// TwinCAT 3 PLC project TcIotOcppServer1Plc
// Title: TwinCAT IoT OCPP Server Sample
// Company: Beckhoff Automation GmbH & Co. KG
// ProjectVersion: 1.0.3.0
// ProgramVersion: 3.1.4026.16
// CompilerDefines: VISU_USEPROPERTYINFO
// libraries:
//   Tc2_EtherCAT, * (Beckhoff Automation GmbH)
//   Tc2_Standard, * (Beckhoff Automation GmbH)
//   Tc2_System, * (Beckhoff Automation GmbH)
//   Tc2_Utilities, * (Beckhoff Automation GmbH)
//   Tc3_Module, * (Beckhoff Automation GmbH)
//   Tc3_OCPP, * (Beckhoff Automation GmbH)
//   VisuDialogs, * (System)
//   VisuSymbols, 4.5.0.0 (System)
// project tree:
//   DUTs/ ST_Connector.TcDUT, ST_VisuStation.TcDUT
//   / GlobalTextList.TcGTLO, PlcTask.TcTTO, Visualization Manager.TcVMO (not stored)
//   GVLs/ VAR_OCPP.TcGVL
//   POUs/ FB_SampledValueMeasurands.TcPOU, FB_Server.TcPOU, FB_Station.TcPOU, MAIN.TcPOU
//   POUs/Helper/ F_ChargePointStatusToString.TcPOU, F_TimeFromString.TcPOU
//   VISUs/ Main_Visu.TcVIS, Measurand.TcVIS, Visu_BootNotification.TcVIS, Visu_Connector.TcVIS, Visu_Station.TcVIS
// real-time tasks:
//   TASK PlcTask: cycle T#1ms, priority 20, ADS port 350

CONFIGURATION TcIotOcppServer1Plc
    RESOURCE PLC ON TwinCAT3
        TASK PlcTask(INTERVAL := T#1ms, PRIORITY := 20);
        PROGRAM MAIN WITH PlcTask : MAIN;
    END_RESOURCE
END_CONFIGURATION

// ---- DUTs/ST_Connector.TcDUT
TYPE ST_Connector :
STRUCT
	sIdTag 				: T_OCPP1_IdToken;
	nReservationId 		: UDINT;
	sStartTime 			: STRING(255);
	sAuthorizationStatus : E_OCPP1_AuthorizationStatus;
	sStopTime 			: STRING(255);
	nTransactionID 		: UDINT; 
	nMeterStart 		: UDINT; // Wh
	nMeterStop 			: UDINT; // Wh 
	sChargpointStatus 	: STRING(31); 
END_STRUCT
END_TYPE

// ---- DUTs/ST_VisuStation.TcDUT
TYPE ST_VisuStation :
STRUCT
	sIdent : T_OCPP_Identity; 
	stBoot : ST_OCPP1_ClientBootInfo; 
	aConnector : ARRAY [0 .. Tc3_Ocpp.Param_OCPP.nConnectorCount] OF ST_Connector; 
END_STRUCT
END_TYPE

// ---- GVLs/VAR_OCPP.TcGVL
{attribute 'qualified_only'}
VAR_GLOBAL
	arrAuthList : ARRAY[1..nAuthListMax] OF ST_OCPP1_AuthorizationData := [
		( sIdTag := '1234abcd', stIdTagInfo := ( eStatus := E_OCPP1_AuthorizationStatus.Accepted ) ),
		( sIdTag := 'B45E00EE', stIdTagInfo := ( eStatus := E_OCPP1_AuthorizationStatus.Accepted ) ),
		( sIdTag := 'A46FF2F1', stIdTagInfo := ( eStatus := E_OCPP1_AuthorizationStatus.Accepted ) )
	];

	stServerParam : ST_OCPP1_ServerParam := (
		//nOID := 16#01010010); 	// ObjectID of the TcIotOcpp Client Object (0 to create a new instance).
		nTaskOID 	:= 0, 			// ObjectId of the Task whose shall execute the client (0 to use I/O Idle Task)
		sHost 		:= '0.0.0.0', 	// Defines the server-address by host-name, domain-name or IP-address.
		nPort 		:= 8080, 		// Defines the server-port.
		sPath 		:= 'ocpp', 		// Defines the server-path.
		eAuthMode 	:= E_OCPP1_AuthenticationMode.Basic, 			// Defines an optional authentication-mode.
		eEncryptionMode := E_OCPP_EncryptionMode.None, 				// Defines an optional encryption mode.
		eEncryptionMode := E_OCPP_EncryptionMode.None, 				// Defines an optional encryption mode.
		eEncryptionProt := E_OCPP_EncryptionProtocol.TLSv1p2, 		// Defines the encryption protocol.
		sCaFile 	:= '%TC_TARGETPATH%\Certificates\CA.crt', 		// Certificate of the certificate authority (CA) as filename (PEM or DER format).
		sCrtFile 	:= '%TC_TARGETPATH%\Certificates\OCPP.crt', 	// Certificate of the server (public key) as filename (PEM or DER format)
		sKeyFile 	:= '%TC_TARGETPATH%\Certificates\OCPP.key', 	// Key of the server (private key) as filename (PEM or DER format).
		eDebugLevel := E_OCPP_DebugLevel.None, 		// Defines the debug level.
		eTraceLevel := TcTraceLevel.tlWarning); 	// Defines the maximum trace level of ADS log messages	
END_VAR

VAR_GLOBAL CONSTANT
	nAuthListMax : UDINT := 3;
	sIdTag : T_OCPP1_IdToken := '1234abcd';
	nReservationId : UDINT := 1234;
END_VAR

// ---- POUs/MAIN.TcPOU
PROGRAM MAIN
VAR
	fbServer : FB_Server(VAR_OCPP.stServerParam);

	fbStation01 : FB_Station('ChargingStation01', '2f20aa42275837973ed8f3726bb2709e0a9e476da9c42da38ac113de818d0dbf', fbServer); // ChargingStation01:abcdef
	fbStation02 : FB_Station('ChargingStation02', '5c55b2828abee6bb262ed0505d53d0baa947e050825ef00e7d3432b722177480', fbServer); // ChargingStation02:abcdef
	//fbStation03 : FB_Station('ChargingStation03', 'f207afc2a29d076265649b050ff3f6449b03dc6d04620e269a17cb31584a4471', fbServer); // ChargingStation03:abcdef
END_VAR

fbStation01.Execute();
fbStation02.Execute();
fbServer.Execute();

END_PROGRAM

// ---- POUs/FB_Server.TcPOU
FUNCTION_BLOCK FB_Server
VAR_OUTPUT
	bValid : BOOL;
END_VAR
VAR
	_fbServer 	: FB_OCPP1_Server(0);
	// receive
	hStationId 	: UDINT;
	hMessageId 	: T_OCPP_MessageId;
	eAction 	: E_OCPP1_Action;
END_VAR

METHOD Execute : BOOL
bValid := _fbServer.bValid;
IF NOT bValid THEN RETURN; END_IF
END_METHOD

METHOD FB_Init : BOOL
VAR_INPUT
	bInitRetains : BOOL; // if TRUE, the retain variables are initialized (warm start / cold start)
	bInCopyCode : BOOL;  // if TRUE, the instance afterwards gets moved into the copy code (online change)

	stParam : REFERENCE TO ST_OCPP1_ServerParam;
END_VAR
IF bInCopyCode THEN RETURN; END_IF

FB_Init := _fbServer.Init(stParam);
END_METHOD

PROPERTY Server : REFERENCE TO FB_OCPP1_Server
GET
Server REF= _fbServer;
END_GET
END_PROPERTY

END_FUNCTION_BLOCK

// ---- POUs/FB_Station.TcPOU
FUNCTION_BLOCK FB_Station
VAR_OUTPUT
	bValid 			: BOOL;
	bOpen			: BOOL;
	bRecv 			: BOOL;
	bReserved 		: BOOL;
	arrCharging 	: ARRAY[0..Param_OCPP.nConnectorCount] OF BOOL; 
	arrStatus 		: ARRAY[0..Param_OCPP.nConnectorCount] OF E_OCPP1_ChargePointStatus;
	arrMeasurands 	: ARRAY[0..Param_OCPP.nConnectorCount] OF FB_SampledValueMeasurands;
END_VAR
VAR
	_fbStation 		: FB_OCPP1_Station('', '', 0);
	_bRecvBoot 		: BOOL := TRUE;
	_bRecvStatus 	: BOOL := TRUE;
	_bRecvMeter 	: BOOL := TRUE;
	_nSendState 	: UDINT;
	_hMessageId 	: T_OCPP_MessageId;
	_eTriggerStatus : E_OCPP1_TriggerMessageStatus;
	
	_stVisu 		: ST_VisuStation;
	_arrRemoteStart	: ARRAY[0..Param_OCPP.nConnectorCount] OF BOOL; 
	_arrRemoteStop	: ARRAY[0..Param_OCPP.nConnectorCount] OF BOOL; 
END_VAR
VAR PERSISTENT
	_nTransactionId		: UDINT;
	_arrTransactionId 	: ARRAY[0..Param_OCPP.nConnectorCount] OF UDINT;
	_arrMeterStart 		: ARRAY[0..Param_OCPP.nConnectorCount] OF UDINT; // [Wh]
	_arrMeterStop 		: ARRAY[0..Param_OCPP.nConnectorCount] OF UDINT; // [Wh]
END_VAR

METHOD ActionHistory : BOOL
VAR_INPUT
	eAction : E_OCPP1_Action;
END_VAR
VAR_STAT
	arrHistory : ARRAY[1..cnCount] OF E_OCPP1_Action;
END_VAR
VAR CONSTANT
	cnCount : UDINT := 100;
END_VAR
MEMMOVE(ADR(arrHistory[2]), ADR(arrHistory[1]), SIZEOF(arrHistory[1]) * (cnCount - 1));
arrHistory[1] := eAction;
END_METHOD

METHOD Authorize : BOOL
VAR_IN_OUT CONSTANT
	sId : T_OCPP1_IdToken;
END_VAR
VAR
	nIdx : UDINT;
END_VAR
FOR nIdx := 1 TO VAR_OCPP.nAuthListMax DO
	IF VAR_OCPP.arrAuthList[nIdx].sIdTag = '' THEN
		RETURN;
	END_IF
	IF VAR_OCPP.arrAuthList[nIdx].sIdTag = sId THEN
		Authorize := (VAR_OCPP.arrAuthList[nIdx].stIdTagInfo.eStatus = E_OCPP1_AuthorizationStatus.Accepted);
		RETURN;
	END_IF
END_FOR
END_METHOD

METHOD Execute : BOOL
VAR_STAT
	hMessageId : T_OCPP_MessageId;
	eAction : E_OCPP1_Action;
	eSendState : E_OCPP1_Action;
	nConnectorId : UDINT; 
END_VAR
VAR
	nIdx : UDINT; 
END_VAR
bValid := _fbStation.bValid;
IF NOT bValid THEN RETURN; END_IF

IF NOT bOpen AND_THEN _fbStation.IsConnected THEN
	bOpen := TRUE;
	bRecv := TRUE;
ELSIF bOpen AND_THEN NOT _fbStation.IsConnected THEN
	bOpen := FALSE;
END_IF

IF _fbStation.PollRequest(eAction => eAction, hMessageId => hMessageId) THEN
	bRecv := TRUE;
	ActionHistory(eAction);
	CASE eAction OF
		E_OCPP1_Action.BootNotification:
			RecvBootNotification();
		E_OCPP1_Action.Heartbeat:
			RecvHeartbeat();
		E_OCPP1_Action.MeterValues:
			RecvMeterValues();
		E_OCPP1_Action.StatusNotification:
			RecvStatusNotification();
		E_OCPP1_Action.Authorize:
			RecvAuthorize();
		E_OCPP1_Action.StartTransaction:
			RecvStartTransaction();
		E_OCPP1_Action.StopTransaction:
			RecvStopTransaction();
		E_OCPP1_Action.DiagnosticsStatusNotification:
			RecvDiagnosticsStatusNotification();
		E_OCPP1_Action.FirmwareStatusNotification:
			RecvFirmwareStatusNotification();
		E_OCPP1_Action.DataTransfer:
			RecvDataTransfer();
		E_OCPP1_Action.SecurityEventNotification:
			RecvSecurityEventNotification();
	ELSE
		_fbStation.RespError(hMessageId, eAction, E_OCPP1_Error.NotImplemented);
	END_CASE
END_IF

// RemoteStart/-Stop from Visu
FOR nIdx := 1 TO Param_OCPP.nConnectorCount DO 
	IF _arrRemoteStart[nIdx] THEN 
		_nSendState := E_OCPP1_Action.RemoteStartTransaction;
		_arrRemoteStart[nIdx] := FALSE; 
		nConnectorId := nIdx; 
	ELSIF _arrRemoteStop[nIdx] THEN 
		_nSendState := E_OCPP1_Action.RemoteStopTransaction;
		_arrRemoteStop[nIdx] := FALSE; 
		nConnectorId := nIdx;
	END_IF
	
	IF nConnectorId = 2 OR NOT bOpen THEN 
		_nSendState := 0;	// Connector not implementet or not connectet
	END_IF
END_FOR

CASE _nSendState OF
	0: // idle
		bRecv := FALSE;
	1:
		IF bRecv THEN
			IF _bRecvBoot THEN
				_bRecvBoot := FALSE;
				_nSendState := 10;
			ELSIF _bRecvStatus THEN
				_bRecvStatus := FALSE;
				_nSendState := 20;
			ELSIF _bRecvMeter THEN
				_bRecvMeter := FALSE;
				_nSendState := 30;
			END_IF
			bRecv := FALSE;
		END_IF
	10: // BootNotification
		IF _fbStation.SendTriggerMessage(eRequestedMessage:= E_OCPP1_MessageTrigger.BootNotification, nConnectorId:= 0, eStatus=> _eTriggerStatus) THEN
			_nSendState := 0;
		END_IF
	20: // StatusNotification
		IF _fbStation.SendTriggerMessage(eRequestedMessage:= E_OCPP1_MessageTrigger.StatusNotification, nConnectorId:= 0, eStatus=> _eTriggerStatus) THEN
			IF _eTriggerStatus = E_OCPP1_TriggerMessageStatus.Accepted THEN
				_nSendState := 21;
			ELSE
				arrStatus[0] := E_OCPP1_ChargePointStatus.Unavailable;
				_nSendState := 0;
			END_IF
		END_IF
	21: // StatusNotification
		IF _fbStation.SendTriggerMessage(eRequestedMessage:= E_OCPP1_MessageTrigger.StatusNotification, nConnectorId:= 1, eStatus=> _eTriggerStatus) THEN
			IF _eTriggerStatus = E_OCPP1_TriggerMessageStatus.Accepted THEN
				_nSendState := 22;
			ELSE
				arrStatus[1] := E_OCPP1_ChargePointStatus.Unavailable;
				_nSendState := 0;
			END_IF
		END_IF
	22: // StatusNotification
		IF _fbStation.SendTriggerMessage(eRequestedMessage:= E_OCPP1_MessageTrigger.StatusNotification, nConnectorId:= 2, eStatus=> _eTriggerStatus) THEN
			IF _eTriggerStatus = E_OCPP1_TriggerMessageStatus.Accepted THEN
				_nSendState := 0;
			ELSE
				arrStatus[2] := E_OCPP1_ChargePointStatus.Unavailable;
				_nSendState := 0;
			END_IF
		END_IF
	30: // MeterValues
		IF _fbStation.SendTriggerMessage(eRequestedMessage:= E_OCPP1_MessageTrigger.MeterValues, nConnectorId:= 0, eStatus=> _eTriggerStatus) THEN
				_nSendState := 31;
		END_IF
	31: // MeterValues
		IF _fbStation.SendTriggerMessage(eRequestedMessage:= E_OCPP1_MessageTrigger.MeterValues, nConnectorId:= 1, eStatus=> _eTriggerStatus) THEN
			IF _eTriggerStatus = E_OCPP1_TriggerMessageStatus.Accepted THEN
				_nSendState := 32;
			ELSE
				_nSendState := 0;
			END_IF
		END_IF
	32: // MeterValues
		IF _fbStation.SendTriggerMessage(eRequestedMessage:= E_OCPP1_MessageTrigger.MeterValues, nConnectorId:= 2, eStatus=> _eTriggerStatus) THEN
			IF _eTriggerStatus = E_OCPP1_TriggerMessageStatus.Accepted THEN
				_nSendState := 0;
			ELSE
				_nSendState := 0;
			END_IF
		END_IF
	E_OCPP1_Action.RemoteStartTransaction:
		SendRemoteStartTransaction();
	E_OCPP1_Action.RemoteStopTransaction:
		SendRemoteStopTransaction();
	E_OCPP1_Action.ChangeAvailability:
		SendChangeAvailability();
	E_OCPP1_Action.ChangeConfiguration:
		SendChangeConfiguration();
	E_OCPP1_Action.GetConfiguration:
		SendGetConfiguration();
	E_OCPP1_Action.UnlockConnector:
		SendUnlockConnector();
	E_OCPP1_Action.ClearCache:
		SendClearCache();
	E_OCPP1_Action.Reset:
		SendReset();
	E_OCPP1_Action.TriggerMessage:
		SendTriggerMessage();
	E_OCPP1_Action.ReserveNow:
		SendReserveNow();
	E_OCPP1_Action.CancelReservation:
		SendCancelReservation();
	E_OCPP1_Action.SetChargingProfile:
		SendChargingProfile();
	E_OCPP1_Action.GetCompositeSchedule:
		SendGetCompositeSchedule();
	E_OCPP1_Action.ClearChargingProfile:
		SendClearChargingProfile();
	E_OCPP1_Action.GetLocalListVersion:
		SendGetLocalListVersion();
	E_OCPP1_Action.SendLocalList:
		SendLocalList();
	E_OCPP1_Action.GetDiagnostics:
		SendGetDiagnostics();
	E_OCPP1_Action.UpdateFirmware:
		SendUpdateFirmware();
	E_OCPP1_Action.DataTransfer:
		SendDataTransfer();
ELSE
	_nSendState := 0;
END_CASE

IF _nSendState = 0 AND eSendState <> 0 THEN
	_nSendState := eSendState;
	eSendState := 0;
END_IF

FOR nIdx := 1 TO Param_OCPP.nConnectorCount DO 
	IF arrCharging[nIdx] THEN 
		_stVisu.aConnector[nIdx].sStopTime := ''; 
		_stVisu.aConnector[nIdx].nMeterStop := 0; 
	ELSE 
		_stVisu.aConnector[nIdx].nMeterStart := _arrMeterStart[nIdx];
		_stVisu.aConnector[nIdx].nMeterStop := _arrMeterStop[nIdx];
	END_IF
	_stVisu.aConnector[nIdx].nTransactionID := _arrTransactionId[nIdx]; 
	_stVisu.aConnector[nIdx].sChargpointStatus := TO_STRING(arrStatus[nIdx]); 
END_FOR
END_METHOD

METHOD FB_Init : BOOL
VAR_INPUT
	bInitRetains : BOOL; // if TRUE, the retain variables are initialized (warm start / cold start)
	bInCopyCode : BOOL;  // if TRUE, the instance afterwards gets moved into the copy code (online change)

	sIdent : T_OCPP_Identity;
	sAuthHash : T_OCPP_Hash;
	fbServer : REFERENCE TO FB_Server;
END_VAR
IF bInCopyCode THEN RETURN; END_IF
_stVisu.sIdent := sIdent; 
FB_Init := _fbStation.Init(sIdent, sAuthHash, fbServer.Server);
END_METHOD

METHOD RecvAuthorize : BOOL
VAR_STAT
	sIdTag : T_OCPP1_IdToken;
END_VAR
IF _fbStation.RecvAuthorize(hMessageId => _hMessageId, sIdTag => sIdTag) THEN
	IF Authorize(sIdTag) THEN
		_fbStation.RespAuthorize(_hMessageId, eStatus := E_OCPP1_AuthorizationStatus.Accepted);
	ELSE
		_fbStation.RespAuthorize(_hMessageId, eStatus := E_OCPP1_AuthorizationStatus.Invalid);
	END_IF
END_IF
END_METHOD

METHOD RecvBootNotification : BOOL
VAR_STAT
	sModel 				: STRING(31);
	sVendor 			: STRING(31);
	sChargeBoxSerial 	: STRING(31);
	sChargePointSerial 	: STRING(31);
	sFirmwareVersion 	: STRING(63);
	sMeterSerial 		: STRING(31);
	sMeterType 			: STRING(31);
END_VAR
IF _fbStation.RecvBootNotification(hMessageId=> _hMessageId,
	sModel=> sModel,
	sVendor=> sVendor,
	sChargeBoxSerial=> sChargeBoxSerial,
	sChargePointSerial=> sChargePointSerial,
	sFirmwareVersion=> sFirmwareVersion,
	sMeterSerial=> sMeterSerial,
	sMeterType=> sMeterType)
THEN
	_fbStation.RespBootNotification(_hMessageId, eStatus := E_OCPP1_RegistrationStatus.Accepted);
			
	_stVisu.stBoot.sChargePointModel 		:= sModel; 				
	_stVisu.stBoot.sChargePointVendor 		:= sVendor; 			
	_stVisu.stBoot.sChargeBoxSerialNumber 	:= sChargeBoxSerial; 	
	_stVisu.stBoot.sChargePointSerialNumber	:= sChargePointSerial; 	
	_stVisu.stBoot.sFirmwareVersion 		:= sFirmwareVersion;	
	_stVisu.stBoot.sMeterSerialNumber 		:= sMeterSerial; 		
	_stVisu.stBoot.sMeterType 				:= sMeterType; 			
	
	_bRecvBoot := FALSE;
END_IF
END_METHOD

METHOD RecvDataTransfer : BOOL
VAR_STAT
	sVendorId : STRING(255);
	sMessageId : STRING(63);
	sData : T_OCPP1_DataTransferData;
END_VAR
IF _fbStation.RecvDataTransfer(hMessageId => _hMessageId,
	sVendorId=> sVendorId,
	sMessageId=> sMessageId,
	sData := sData)
THEN
	IF sVendorId <> 'Beckhoff Automation' THEN
		_fbStation.RespDataTransfer(_hMessageId, eStatus := E_OCPP1_DataTransferStatus.UnknownVendorId);
	ELSIF sMessageId <> 'DataTransfer' THEN
		_fbStation.RespDataTransfer(_hMessageId, eStatus := E_OCPP1_DataTransferStatus.UnknownMessageId);
	ELSE
		_fbStation.RespDataTransfer(_hMessageId, eStatus := E_OCPP1_DataTransferStatus.Accepted);
	END_IF
END_IF
END_METHOD

METHOD RecvDiagnosticsStatusNotification : BOOL
IF _fbStation.RecvDiagnosticsStatusNotification(hMessageId => _hMessageId) THEN
	_fbStation.RespDiagnosticsStatusNotification(_hMessageId);
END_IF
END_METHOD

METHOD RecvFirmwareStatusNotification : BOOL
IF _fbStation.RecvFirmwareStatusNotification(hMessageId => _hMessageId) THEN
	_fbStation.RespFirmwareStatusNotification(_hMessageId);
END_IF
END_METHOD

METHOD RecvHeartbeat : BOOL
VAR_STAT
	nHeartbeats : UDINT;
END_VAR
IF _fbStation.RecvHeartbeat(hMessageId => _hMessageId) THEN
	nHeartbeats := nHeartbeats + 1;
	_fbStation.RespHeartbeat(_hMessageId);
END_IF
END_METHOD

METHOD RecvMeterValues : BOOL
VAR_STAT
	nConnectorId : UDINT;
	nTransactionId : UDINT;
	nSampleCount : UDINT;
	arrSampleValues : ARRAY[1..Param_OCPP.nSampledValuesMax] OF ST_OCPP1_SampledValue;
END_VAR
IF _fbStation.RecvMeterValue(
	hMessageId => _hMessageId,
	nConnectorId => nConnectorId,
	nTransactionId => nTransactionId,
	nSampleCount => nSampleCount,
	aSampleValues := arrSampleValues)
THEN
	IF nConnectorId >= 0 AND nConnectorId <= Param_OCPP.nConnectorCount THEN
		arrMeasurands[nConnectorId].Update(arrSampleValues);
	END_IF
	_fbStation.RespMeterValue(_hMessageId);
	_bRecvMeter := FALSE;
END_IF
END_METHOD

METHOD RecvSecurityEventNotification : BOOL
VAR_STAT
	nTimestamp : ULINT;
	sType : STRING(63);
	sInfo : STRING(256);
END_VAR
IF _fbStation.RecvSecurityEventNotification(hMessageId => _hMessageId,
	nTimestamp => nTimestamp,
	sType => sType,
	sInfo => sInfo)
THEN
	_fbStation.RespSecurityEventNotification(_hMessageId);
END_IF
END_METHOD

METHOD RecvStartTransaction : BOOL
VAR_STAT
	sIdTag : T_OCPP1_IdToken;
	nConnectorId : UDINT;
	nMeterStart : UDINT;
	nReservationId : UDINT;
	nTimestamp : ULINT;
END_VAR
IF _fbStation.RecvStartTransaction(hMessageId => _hMessageId,
	sIdTag => sIdTag,
	nConnectorId => nConnectorId,
	nMeterStart => nMeterStart,
	nReservationId => nReservationId,
	nTimestamp => nTimestamp)
THEN


	_stVisu.aConnector[nConnectorId].sIdTag := sIdTag; 
	
	IF Authorize(sIdTag) THEN
		IF nConnectorId >= 1 AND nConnectorId <= Param_OCPP.nConnectorCount THEN
			_nTransactionId := _nTransactionId + 1;
			_arrTransactionId[nConnectorId] := _nTransactionId;
			_arrMeterStart[nConnectorId] := nMeterStart;
			_fbStation.RespStartTransaction(_hMessageId, eStatus := E_OCPP1_AuthorizationStatus.Accepted, nTransactionId := _nTransactionId);
			arrCharging[nConnectorId] := TRUE; 
			_stVisu.aConnector[nConnectorId].nReservationId := nReservationId; 
			_stVisu.aConnector[nConnectorId].sStartTime := TO_STRING(FILETIME64_TO_DT(nTimestamp)); 			
			_stVisu.aConnector[nConnectorId].sAuthorizationStatus := E_OCPP1_AuthorizationStatus.Accepted; 
			RETURN;
		END_IF
	END_IF
	_fbStation.RespStartTransaction(_hMessageId, eStatus := E_OCPP1_AuthorizationStatus.Invalid, nTransactionId := 0);
END_IF
END_METHOD

METHOD RecvStatusNotification : BOOL
VAR_STAT
	nConnectorId : UDINT;
	eError : E_OCPP1_ChargePointError;
	eStatus : E_OCPP1_ChargePointStatus;
	nTimestamp : ULINT := 0;
	sInfo : STRING(63) := '';
	sVendorError : STRING(63) := '';
	sVendorId : STRING(255) := '';
END_VAR
IF _fbStation.RecvStatusNotification(hMessageId => _hMessageId,
	nConnectorId => nConnectorId,
	eError => eError,
	eStatus => eStatus,
	nTimestamp => nTimestamp,
	sInfo => sInfo,
	sVendorError => sVendorError,
	sVendorId => sVendorId)
THEN
	IF nConnectorId >= 0 AND nConnectorId <= Param_OCPP.nConnectorCount THEN
		arrStatus[nConnectorId] := eStatus;
		StatusHistory(nConnectorId, eStatus);
		arrCharging[nConnectorId] := (eStatus = E_OCPP1_ChargePointStatus.Charging);
		bReserved := (eStatus = E_OCPP1_ChargePointStatus.Reserved);
	END_IF
	_fbStation.RespStatusNotification(_hMessageId);
	_bRecvStatus := FALSE;
END_IF
END_METHOD

METHOD RecvStopTransaction : BOOL
VAR_STAT
	sIdTag : T_OCPP1_IdToken;
	nTransactionId : UDINT;
	nConnectorId : UDINT;
	nMeterStop : UDINT;
	nTimestamp : ULINT;
	eReason : E_OCPP1_Reason;
END_VAR
VAR
	nIdx : UDINT;
END_VAR
IF _fbStation.RecvStopTransaction(hMessageId => _hMessageId,
	sIdTag => sIdTag,
	nTransactionId => nTransactionId,
	nConnectorId => nConnectorId,
	nMeterStop => nMeterStop,
	nTimestamp => nTimestamp,
	eReason => eReason)
THEN
	IF sIdTag = '' OR_ELSE Authorize(sIdTag) THEN
		IF nConnectorId >= 1 AND nConnectorId <= Param_OCPP.nConnectorCount THEN
			_arrTransactionId[nConnectorId] := 0;
			_arrMeterStop[nConnectorId] := nMeterStop;
			_fbStation.RespStopTransaction(_hMessageId, eStatus := E_OCPP1_AuthorizationStatus.Accepted);
			arrCharging[nConnectorId] := FALSE; 
			
			_stVisu.aConnector[nConnectorId].sStopTime := TO_STRING(FILETIME64_TO_DT(nTimestamp));
			RETURN;
		END_IF
		FOR nIdx := 1 TO Param_OCPP.nConnectorCount DO
			IF _arrTransactionId[nIdx] = nTransactionId THEN
				_arrTransactionId[nIdx] := 0;
				_arrMeterStop[nIdx] := nMeterStop;
				_fbStation.RespStopTransaction(_hMessageId, eStatus := E_OCPP1_AuthorizationStatus.Accepted);
				arrCharging[nIdx] := FALSE; 
				
				_stVisu.aConnector[nIdx].sStopTime := TO_STRING(FILETIME64_TO_DT(nTimestamp)); 
				RETURN;
 			END_IF
		END_FOR
	END_IF
	_fbStation.RespStopTransaction(_hMessageId, eStatus := E_OCPP1_AuthorizationStatus.Invalid);
END_IF
END_METHOD

METHOD SendCancelReservation : BOOL
VAR_STAT
	nReservationId : UDINT := VAR_OCPP.nReservationId;
	eStatus : E_OCPP1_CancelReservationStatus;
END_VAR
IF _fbStation.SendCancelReservation(nReservationId:= nReservationId, eStatus=> eStatus) THEN
	bReserved := (eStatus <> E_OCPP1_CancelReservationStatus.Accepted);
	_nSendState := 0;
END_IF
END_METHOD

METHOD SendChangeAvailability : BOOL
VAR_STAT
	nConnectorId : UDINT := 1;
	eType : E_OCPP1_AvailabilityType;
	eStatus : E_OCPP1_AvailabilityStatus;
END_VAR
IF eType = E_OCPP1_AvailabilityType.None THEN
	IF arrStatus[1] = E_OCPP1_ChargePointStatus.Unavailable THEN
		eType := E_OCPP1_AvailabilityType.Operative;
	ELSE
		eType := E_OCPP1_AvailabilityType.Inoperative;
	END_IF
END_IF
IF _fbStation.SendChangeAvailability(nConnectorId := nConnectorId, eType := eType, eStatus => eStatus) THEN
	eType := E_OCPP1_AvailabilityType.None;
	_nSendState := 0;
END_IF
END_METHOD

METHOD SendChangeConfiguration : BOOL
VAR_STAT
	sKey : T_OCPP1_ConfigKey;
	sValue : T_OCPP1_ConfigValue;
	eStatus : E_OCPP1_ConfigurationStatus;
END_VAR
IF sKey = '' THEN
	eStatus := E_OCPP1_ConfigurationStatus.Rejected;
	RETURN;
END_IF
IF _fbStation.SendChangeConfiguration(sKey:= sKey, sValue:= sValue, eStatus=> eStatus) THEN
	_nSendState := 0;
END_IF
END_METHOD

METHOD SendChargingProfile : BOOL
VAR_STAT
	nConnectorId : UDINT := 1;
	mChargingProfile : ST_OCPP1_ChargingProfileMax;
	eStatus : E_OCPP1_ChargingProfileStatus;
END_VAR
IF mChargingProfile.nProfileId = 0 THEN
	mChargingProfile.nProfileId := 1;
	mChargingProfile.nTransactionId := 0;
	mChargingProfile.nStackLevel := 1;
	mChargingProfile.eProfilePurpose := E_OCPP1_ChargingProfilePurposeType.TxDefaultProfile;
	mChargingProfile.eProfileKind :=	E_OCPP1_ChargingProfileKindType.Relative;
	mChargingProfile.eRecurrencyKind := E_OCPP1_RecurrencyKindType.None;
	mChargingProfile.nValidFrom := 0;
	mChargingProfile.nValidTo := 0;
	mChargingProfile.mSchedule.nStart := 0;
	mChargingProfile.mSchedule.nDuration := 0;
	mChargingProfile.mSchedule.eRateUnit := E_OCPP1_ChargingRateUnitType.A;
	mChargingProfile.mSchedule.fRateMin := 0.0;
	mChargingProfile.mSchedule.nPeriodCount := 6;
	mChargingProfile.mSchedule.aPeriods[1].nStart := 0;
	mChargingProfile.mSchedule.aPeriods[1].fLimit := 2.0; // 2A => 1.380W
	mChargingProfile.mSchedule.aPeriods[2].nStart := 60;
	mChargingProfile.mSchedule.aPeriods[2].fLimit := 4.0; // 4A => 2.760W
	mChargingProfile.mSchedule.aPeriods[3].nStart := 120;
	mChargingProfile.mSchedule.aPeriods[3].fLimit := 6.0; // 6A => 4.140W
	mChargingProfile.mSchedule.aPeriods[4].nStart := 180;
	mChargingProfile.mSchedule.aPeriods[4].fLimit := 8.0; // 8A => 5.520W
	mChargingProfile.mSchedule.aPeriods[5].nStart := 240;
	mChargingProfile.mSchedule.aPeriods[5].fLimit := 10.0; // 10A => 6.900W
	mChargingProfile.mSchedule.aPeriods[6].nStart := 300;
	mChargingProfile.mSchedule.aPeriods[6].fLimit := 16.0; // 16A => 11.040W
END_IF
IF _fbStation.SendChargingProfile(nConnectorId:= nConnectorId, mChargingProfile:= mChargingProfile, eStatus=> eStatus) THEN
	_nSendState := 0;
END_IF
END_METHOD

METHOD SendClearCache : BOOL
VAR_STAT
	eStatus : E_OCPP1_ClearCacheStatus;
END_VAR
IF _fbStation.SendClearCache(eStatus => eStatus) THEN
	_nSendState := 0;
END_IF
END_METHOD

METHOD SendClearChargingProfile : BOOL
VAR_STAT
	nProfileId : UDINT := 1;
	nConnectorId : UDINT := 1;
	eChargingProfilePurpose : E_OCPP1_ChargingProfilePurposeType := E_OCPP1_ChargingProfilePurposeType.None;
	nStackLevel : UDINT := 0;
	eStatus : E_OCPP1_ClearChargingProfileStatus;
END_VAR
IF _fbStation.SendClearChargingProfile(
	nProfileId:= nProfileId,
	nConnectorId:= nConnectorId,
	eChargingProfilePurpose:= eChargingProfilePurpose,
	nStackLevel:= nStackLevel,
	eStatus=> eStatus)
THEN
	_nSendState := 0;
END_IF
END_METHOD

METHOD SendDataTransfer : BOOL
VAR_STAT
	sVendorId : STRING(255) := 'Beckhoff Automation'; 
	sMessageId : STRING(63) := 'DataTransfer'; 
	sData : T_OCPP1_DataTransferData := '{"Vendor":"Beckhoff Automation","Message":"DataTransfer","Data":"This is a test message"}'; 
	eStatus : E_OCPP1_DataTransferStatus;
END_VAR
IF _fbStation.SendDataTransfer(sVendorId, sMessageId, sData, eStatus => eStatus) THEN
	_nSendState := 0;
END_IF
END_METHOD

METHOD SendGetCompositeSchedule : BOOL
VAR_STAT
	nConnectorId : UDINT := 1;
	nDuration : UDINT := 24 * 3600;
	eChargingRateUnit : E_OCPP1_ChargingRateUnitType := E_OCPP1_ChargingRateUnitType.A;
	eStatus : E_OCPP1_GetCompositeScheduleStatus;
	nConnectorIdRes : UDINT;
	nScheduleStart : ULINT := 0;
	mChargingSchedule : ST_OCPP1_ChargingScheduleMax;
END_VAR
IF _fbStation.SendGetCompositeSchedule(
	nConnectorId:= nConnectorId,
	nDuration:= nDuration,
	eChargingRateUnit := eChargingRateUnit,
	eStatus=> eStatus,
	nConnectorIdRes => nConnectorIdRes,
	nScheduleStart => nScheduleStart,
	mChargingSchedule=> mChargingSchedule)
THEN
	_nSendState := 0;
END_IF
END_METHOD

METHOD SendGetConfiguration : BOOL
VAR_STAT
	nKeysCount : UDINT := 0;
	nUnknownCount : UDINT := 0;
	arrKeys : ARRAY[1..Param_OCPP.nConfigKeysMax] OF ST_OCPP1_ConfigKeyValue;
END_VAR
IF _fbStation.SendGetConfiguration(nKeysCount => nKeysCount, nUnknownCount => nUnknownCount, aKeys:= arrKeys) THEN
	_nSendState := 0;
END_IF
END_METHOD

METHOD SendGetDiagnostics : BOOL
VAR_STAT
	sLocation : STRING(255) := 'dummy.txt';
	nRetries : UDINT := 3;
	nRetryInterval : UDINT := 60;
	nStartTime : ULINT;
	nStopTime : ULINT;
	sFileName : STRING(255); // Optional. This contains the name of the file with diagnostic information that will be uploaded.
END_VAR
IF _fbStation.SendGetDiagnostics(
	sLocation:= sLocation,
	nRetries:= nRetries,
	nRetryInterval:= nRetryInterval,
	nStartTime:= nStartTime,
	nStopTime:= nStopTime,
	sFileName=> sFileName)
THEN
	_nSendState := 0;
END_IF
END_METHOD

METHOD SendGetLocalListVersion : BOOL
VAR_STAT
	nListVersion : UDINT;
END_VAR
IF _fbStation.SendGetLocalListVersion(nListVersion => nListVersion) THEN
	_nSendState := 0;
END_IF
END_METHOD

METHOD SendLocalList : BOOL
VAR_STAT
	nListVersion : UDINT := 1;
	eUpdateType : E_OCPP1_UpdateType := E_OCPP1_UpdateType.Full;
	eStatus : E_OCPP1_UpdateStatus;
END_VAR
IF _fbStation.SendLocalList(
	nListVersion:= nListVersion,
	eUpdateType:= eUpdateType,
	nAuthCount:= VAR_OCPP.nAuthListMax,
	aAuthList:= VAR_OCPP.arrAuthList,
	eStatus=> eStatus)
THEN
	_nSendState := 0;
END_IF
END_METHOD

METHOD SendRemoteStartTransaction : BOOL
VAR_INPUT
	nConnectorId : UDINT := 1;
END_VAR
VAR_STAT
	sIdToken : T_OCPP1_IdToken := VAR_OCPP.sIdTag;
	eStatus : E_OCPP1_RemoteStartStopStatus; // Required. Status indicating whether Charge Point accepts the request to start a transaction.
END_VAR
IF _fbStation.SendRemoteStartTransaction(nConnectorId := nConnectorId, sIdToken := sIdToken, eStatus => eStatus) THEN
	arrCharging[nConnectorId] := (eStatus = E_OCPP1_RemoteStartStopStatus.Accepted);
	_nSendState := 0;
END_IF
END_METHOD

METHOD SendRemoteStopTransaction : BOOL
VAR_INPUT
	nConnectorId : UDINT := 1;
END_VAR
VAR_STAT
	nTransactionId : UDINT;
	eStatus : E_OCPP1_RemoteStartStopStatus;
END_VAR
IF nTransactionId = 0 THEN
	nTransactionId := _arrTransactionId[nConnectorId];
END_IF
IF _fbStation.SendRemoteStopTransaction(nTransactionId := nTransactionId, eStatus => eStatus) THEN
	nTransactionId := 0;
	arrCharging[nConnectorId] := (eStatus <> E_OCPP1_RemoteStartStopStatus.Accepted);
	_nSendState := 0;
END_IF
END_METHOD

METHOD SendReserveNow : BOOL
VAR_STAT
	nConnectorId : UDINT := 1;
	nExpiryDate : ULINT;
	sIdTag : T_OCPP1_IdToken := VAR_OCPP.sIdTag;
	nReservationId : UDINT := VAR_OCPP.nReservationId;
	eStatus : E_OCPP1_ReservationStatus;
END_VAR
IF nExpiryDate = 0 THEN
	nExpiryDate := F_GetSystemTime() + 3600 * 10000000;
END_IF
IF _fbStation.SendReserveNow(
	nConnectorId:= nConnectorId,
	nExpiryDate:= nExpiryDate,
	sIdTag:= sIdTag,
	sParentIdTag:= '',
	nReservationId:= nReservationId,
	eStatus=> eStatus)
THEN
	bReserved := (eStatus = E_OCPP1_ReservationStatus.Accepted);
	_nSendState := 0;
END_IF
END_METHOD

METHOD SendReset : BOOL
VAR_STAT
	eType : E_OCPP1_ResetType := E_OCPP1_ResetType.Hard;
	eStatus : E_OCPP1_ResetStatus;
END_VAR
IF _fbStation.SendReset(eType := eType, eStatus => eStatus) THEN
	_nSendState := 0;
END_IF
END_METHOD

METHOD SendTriggerMessage : BOOL
VAR_STAT
	eRequestedMessage : E_OCPP1_MessageTrigger := E_OCPP1_MessageTrigger.Heartbeat;
	nConnectorId : UDINT := 0;
	eStatus : E_OCPP1_TriggerMessageStatus;
END_VAR
IF _fbStation.SendTriggerMessage(eRequestedMessage:= eRequestedMessage, nConnectorId:= nConnectorId, eStatus=> eStatus) THEN
	_nSendState := 0;
END_IF
END_METHOD

METHOD SendUnlockConnector : BOOL
VAR_STAT
	nConnectorId : UDINT := 1;
	eStatus : E_OCPP1_UnlockStatus;
END_VAR
IF _fbStation.SendUnlockConnector(nConnectorId := nConnectorId, eStatus => eStatus) THEN
	_nSendState := 0;
END_IF
END_METHOD

METHOD SendUpdateFirmware : BOOL
VAR_STAT
	sLocation : STRING(255);
	nRetries : UDINT := 3;
	nRetryInterval : UDINT := 60;
	nRetrieveDate : ULINT;
END_VAR
IF nRetrieveDate = 0 THEN
	nRetrieveDate := F_GetSystemTime();
END_IF
IF _fbStation.SendUpdateFirmware(
	sLocation := sLocation,
	nRetries := nRetries,
	nRetryInterval := nRetryInterval,
	nRetrieveDate := nRetrieveDate)
THEN
	_nSendState := 0;
END_IF
END_METHOD

METHOD StatusHistory : BOOL
VAR_INPUT
	nConnectorId : UDINT;
	eStatus : E_OCPP1_ChargePointStatus;
END_VAR
VAR
	arrHistory : REFERENCE TO ARRAY[1..cnCount] OF E_OCPP1_ChargePointStatus;;
END_VAR
VAR_STAT
	arrConnectorHistory : ARRAY[0..Param_OCPP.nConnectorCount] OF ARRAY[1..cnCount] OF E_OCPP1_ChargePointStatus;
END_VAR
VAR CONSTANT
	cnCount : UDINT := 100;
END_VAR
IF nConnectorId <= Param_OCPP.nConnectorCount THEN
	arrHistory REF= arrConnectorHistory[nConnectorId];
	MEMMOVE(ADR(arrHistory[2]), ADR(arrHistory[1]), SIZEOF(arrHistory[1]) * (cnCount - 1));
	arrHistory[1] := eStatus;
END_IF
END_METHOD

METHOD TrigReserveCancel : BOOL
IF _nSendState = 0 THEN
	_nSendState := E_OCPP1_Action.CancelReservation;
	TrigReserveCancel := TRUE;
END_IF
END_METHOD

METHOD TrigReserveNow : BOOL
IF _nSendState = 0 THEN
	_nSendState := E_OCPP1_Action.ReserveNow;
	TrigReserveNow := TRUE;
END_IF
END_METHOD

METHOD TrigStartTransaction : BOOL
IF _nSendState = 0 THEN
	_nSendState := E_OCPP1_Action.RemoteStartTransaction;
	TrigStartTransaction := TRUE;
END_IF
END_METHOD

METHOD TrigStopTransaction : BOOL
IF _nSendState = 0 THEN
	_nSendState := E_OCPP1_Action.RemoteStopTransaction;
	TrigStopTransaction := TRUE;
END_IF
END_METHOD

END_FUNCTION_BLOCK

// ---- POUs/FB_SampledValueMeasurands.TcPOU
FUNCTION_BLOCK FB_SampledValueMeasurands
VAR_OUTPUT
	nUpdateTimestamp : ULINT; // Last timestamp for measured value(s).
	sUpdateTimestamp : STRING(23); // Last timestamp for measured value(s).
	fCurrentExport : REAL := -1.0; // [A] Instantaneous current flow from EV
	fCurrentImport : REAL := -1.0; // [A] Instantaneous current flow to EV
	fCurrentImportL1 : REAL := -1.0; // [A] Instantaneous current flow to EV
	fCurrentImportL2 : REAL := -1.0; // [A] Instantaneous current flow to EV
	fCurrentImportL3 : REAL := -1.0; // [A] Instantaneous current flow to EV
	fCurrentOffered : REAL := -1.0; // [A] Maximum current offered to EV
	fEnergyActiveExportRegister : REAL := -1.0; // [kWh] Numerical value read from the "active electrical energy" (Wh or kWh) register of the (most authoritative) electrical meter measuring energy exported (to the grid).
	fEnergyActiveImportRegister : REAL := -1.0; // [kWh] Numerical value read from the "active electrical energy" (Wh or kWh) register of the (most authoritative) electrical meter measuring energy imported (from the grid supply).
	fEnergyReactiveExportRegister : REAL := -1.0; // [kVARh] Numerical value read from the "reactive electrical energy" (VARh or kVARh) register of the (most authoritative) electrical meter measuring energy exported (to the grid).
	fEnergyReactiveImportRegister : REAL := -1.0; // [kVARh] Numerical value read from the "reactive electrical energy" (VARh or kVARh) register of the (most authoritative) electrical meter measuring energy imported (from the grid supply).
	fEnergyActiveExportInterval : REAL := -1.0; // [kWh] Absolute amount of "active electrical energy" (Wh or kWh) exported (to the grid) during an associated time "interval".
	fEnergyActiveImportInterval : REAL := -1.0; // [kWh] Absolute amount of "active electrical energy" (Wh or kWh) imported(from the grid supply) during an associated time "interval".
	fEnergyReactiveExportInterval : REAL := -1.0; // [kVARh] Absolute amount of "reactive electrical energy" (VARh or kVARh) exported (to the grid) during an associated time "interval".
	fEnergyReactiveImportInterval : REAL := -1.0; // [kVARh] Absolute amount of "reactive electrical energy" (VARh or kVARh) imported (from the grid supply) during an associated time "interval".
	fFrequency : REAL := -1.0; // [Hz] Instantaneous reading of powerline frequency.
	fPowerActiveExport : REAL := -1.0; // [kW] Instantaneous active power exported by EV. (W or kW)
	fPowerActiveImport : REAL := -1.0; // [kW] Instantaneous active power imported by EV. (W or kW)
	fPowerOffered : REAL := -1.0; // [kW] Maximum power offered to EV
	fPowerFactor : REAL := -1.0; // Instantaneous power factor of total energy flow
	fPowerReactiveExport : REAL := -1.0; // [VAR] Instantaneous reactive power exported by EV. (var or kvar)
	fPowerReactiveImport : REAL := -1.0; // [VAR] Instantaneous reactive power imported by EV. (var or kvar)
	fFanSpeed : REAL := -1.0; // [r/m] Fan speed in RPM
	fStateOfCharge : REAL := -1.0; // [%] State of charge of charging vehicle in percentage
	fTemperature : REAL := -1.0; // [°C] Temperature reading inside Charge Point.
	fVoltage : REAL := -1.0; // [V] Instantaneous AC RMS supply voltage
	fVoltageL1N : REAL := -1.0; // [V] Instantaneous AC RMS supply voltage
	fVoltageL2N : REAL := -1.0; // [V] Instantaneous AC RMS supply voltage
	fVoltageL3N : REAL := -1.0; // [V] Instantaneous AC RMS supply voltage
END_VAR
VAR
	mErrorValue : ST_OCPP1_SampledValue;
END_VAR

METHOD Update : BOOL
VAR_IN_OUT CONSTANT
	arrSampleValues : ARRAY[*] OF ST_OCPP1_SampledValue;
END_VAR
VAR
	nIdx : DINT;
END_VAR
FOR nIdx := LOWER_BOUND(arrSampleValues,1) TO UPPER_BOUND(arrSampleValues,1) DO
	IF arrSampleValues[nIdx].nTimestamp > nUpdateTimestamp THEN
		nUpdateTimestamp := arrSampleValues[nIdx].nTimestamp;
		sUpdateTimestamp := DCTIME64_TO_STRING(FILETIME64_TO_DCTIME64(nUpdateTimestamp));
	END_IF
    UpdateRawValue(arrSampleValues[nIdx]);
END_FOR
END_METHOD

METHOD UpdateRawValue : BOOL
VAR_IN_OUT CONSTANT
	mValue : ST_OCPP1_SampledValue;
END_VAR
VAR
	fValue : REAL;
END_VAR
VAR CONSTANT
	cfOneKilo : REAL := 0.001;
	cfOneThird : REAL := 1.0 / 3.0;
END_VAR
fValue := LREAL_TO_REAL(mValue.fValue);
IF mValue.ePhase = E_OCPP1_Phase.None THEN
	CASE mValue.eMeasurand OF
		E_OCPP1_Measurand.CurrentExport:
			IF mValue.eUnit = E_OCPP1_Unit.A THEN
				fCurrentExport := fValue;
			ELSE
				mErrorValue := mValue;
			END_IF
		E_OCPP1_Measurand.CurrentImport:
			IF mValue.eUnit = E_OCPP1_Unit.A THEN
				fCurrentImport := fValue;
			ELSE
				mErrorValue := mValue;
			END_IF
		E_OCPP1_Measurand.CurrentOffered:
			IF mValue.eUnit = E_OCPP1_Unit.A THEN
				fCurrentOffered := fValue;
			ELSE
				mErrorValue := mValue;
			END_IF
		E_OCPP1_Measurand.EnergyActiveExportRegister:
			IF mValue.eUnit = E_OCPP1_Unit.Wh THEN
				fEnergyActiveExportRegister := fValue * cfOneKilo;
			ELSIF mValue.eUnit = E_OCPP1_Unit.kWh THEN
				fEnergyActiveExportRegister := fValue;
			ELSE
				mErrorValue := mValue;
			END_IF
		E_OCPP1_Measurand.EnergyActiveImportRegister:
			IF mValue.eUnit = E_OCPP1_Unit.Wh THEN
				fEnergyActiveImportRegister := fValue * cfOneKilo;
			ELSIF mValue.eUnit = E_OCPP1_Unit.kWh THEN
				fEnergyActiveImportRegister := fValue;
			ELSE
				mErrorValue := mValue;
			END_IF
		E_OCPP1_Measurand.EnergyReactiveExportRegister:
			IF mValue.eUnit = E_OCPP1_Unit.VARh THEN
				fEnergyReactiveExportRegister := fValue * cfOneKilo;
			ELSIF mValue.eUnit = E_OCPP1_Unit.kVARh THEN
				fEnergyReactiveExportRegister := fValue;
			ELSE
				mErrorValue := mValue;
			END_IF
		E_OCPP1_Measurand.EnergyReactiveImportRegister:
			IF mValue.eUnit = E_OCPP1_Unit.VARh THEN
				fEnergyReactiveImportRegister := fValue * cfOneKilo;
			ELSIF mValue.eUnit = E_OCPP1_Unit.kVARh THEN
				fEnergyReactiveImportRegister := fValue;
			ELSE
				mErrorValue := mValue;
			END_IF
		E_OCPP1_Measurand.EnergyActiveExportInterval:
			IF mValue.eUnit = E_OCPP1_Unit.Wh THEN
				fEnergyActiveExportInterval := fValue * cfOneKilo;
			ELSIF mValue.eUnit = E_OCPP1_Unit.kWh THEN
				fEnergyActiveExportInterval := fValue;
			ELSE
				mErrorValue := mValue;
			END_IF
		E_OCPP1_Measurand.EnergyActiveImportInterval:
			IF mValue.eUnit = E_OCPP1_Unit.Wh THEN
				fEnergyActiveImportInterval := fValue * cfOneKilo;
			ELSIF mValue.eUnit = E_OCPP1_Unit.kWh THEN
				fEnergyActiveImportInterval := fValue;
			ELSE
				mErrorValue := mValue;
			END_IF
		E_OCPP1_Measurand.EnergyReactiveExportInterval:
			IF mValue.eUnit = E_OCPP1_Unit.VARh THEN
				fEnergyReactiveExportInterval := fValue * cfOneKilo;
			ELSIF mValue.eUnit = E_OCPP1_Unit.kVARh THEN
				fEnergyReactiveExportInterval := fValue;
			ELSE
				mErrorValue := mValue;
			END_IF
		E_OCPP1_Measurand.EnergyReactiveImportInterval:
			IF mValue.eUnit = E_OCPP1_Unit.VARh THEN
				fEnergyReactiveImportInterval := fValue * cfOneKilo;
			ELSIF mValue.eUnit = E_OCPP1_Unit.kVARh THEN
				fEnergyReactiveImportInterval := fValue;
			ELSE
				mErrorValue := mValue;
			END_IF
		E_OCPP1_Measurand.Frequency:
			IF mValue.eUnit = E_OCPP1_Unit.None THEN
				fFrequency := fValue;
			ELSE
				mErrorValue := mValue;
			END_IF
		E_OCPP1_Measurand.PowerActiveExport:
			IF mValue.eUnit = E_OCPP1_Unit.W THEN
				fPowerActiveExport := fValue * cfOneKilo;
			ELSIF mValue.eUnit = E_OCPP1_Unit.kW THEN
				fPowerActiveExport := fValue;
			ELSE
				mErrorValue := mValue;
			END_IF
		E_OCPP1_Measurand.PowerActiveImport:
			IF mValue.eUnit = E_OCPP1_Unit.W THEN
				fPowerActiveImport := fValue * cfOneKilo;
			ELSIF mValue.eUnit = E_OCPP1_Unit.kW THEN
				fPowerActiveImport := fValue;
			ELSE
				mErrorValue := mValue;
			END_IF
		E_OCPP1_Measurand.PowerOffered:
			IF mValue.eUnit = E_OCPP1_Unit.W THEN
				fPowerOffered := fValue * cfOneKilo;
			ELSIF mValue.eUnit = E_OCPP1_Unit.kW THEN
				fPowerOffered := fValue;
			ELSE
				mErrorValue := mValue;
			END_IF
		E_OCPP1_Measurand.PowerFactor:
			IF mValue.eUnit = E_OCPP1_Unit.None THEN
				fPowerFactor := fValue;
			ELSE
				mErrorValue := mValue;
			END_IF
		E_OCPP1_Measurand.PowerReactiveExport:
			IF mValue.eUnit = E_OCPP1_Unit.Vars THEN
				fPowerReactiveExport := fValue;
			ELSE
				mErrorValue := mValue;
			END_IF
		E_OCPP1_Measurand.PowerReactiveImport:
			IF mValue.eUnit = E_OCPP1_Unit.Vars THEN
				fPowerReactiveImport := fValue;
			ELSE
				mErrorValue := mValue;
			END_IF
		E_OCPP1_Measurand.RPM:
			IF mValue.eUnit = E_OCPP1_Unit.None THEN
				fFanSpeed := fValue;
			ELSE
				mErrorValue := mValue;
			END_IF
		E_OCPP1_Measurand.SoC:
			IF mValue.eUnit = E_OCPP1_Unit.Percent THEN
				fStateOfCharge := fValue;
			ELSE
				mErrorValue := mValue;
			END_IF
		E_OCPP1_Measurand.Temperature:
			IF mValue.eUnit = E_OCPP1_Unit.Celsius THEN
				fTemperature := fValue;
			ELSE
				mErrorValue := mValue;
			END_IF
		E_OCPP1_Measurand.Voltage:
			IF mValue.eUnit = E_OCPP1_Unit.V THEN
				fVoltage := fValue;
			ELSE
				mErrorValue := mValue;
			END_IF
	ELSE
		mErrorValue := mValue;
	END_CASE
ELSE
	CASE mValue.eMeasurand OF
		E_OCPP1_Measurand.CurrentImport:
			IF mValue.eUnit = E_OCPP1_Unit.A THEN
				IF mValue.ePhase = E_OCPP1_Phase.None THEN
					fCurrentImport := fValue;
				ELSE
					CASE mValue.ePhase OF
						E_OCPP1_Phase.L1: fCurrentImportL1 := fValue;
						E_OCPP1_Phase.L2: fCurrentImportL2 := fValue;
						E_OCPP1_Phase.L3: fCurrentImportL3 := fValue;
					ELSE
						mErrorValue := mValue;
					END_CASE
					IF fCurrentImportL1 >= 0 AND fCurrentImportL2 >= 0 AND fCurrentImportL3 >= 0 THEN
						fCurrentImport := (fCurrentImportL1 + fCurrentImportL2 + fCurrentImportL3);
					END_IF
				END_IF
			ELSE
				mErrorValue := mValue;
			END_IF
		E_OCPP1_Measurand.Voltage:
			IF mValue.eUnit = E_OCPP1_Unit.V THEN
				IF mValue.ePhase = E_OCPP1_Phase.None THEN
					fVoltage := fValue;
				ELSE
					CASE mValue.ePhase OF
						E_OCPP1_Phase.L1N: fVoltageL1N := fValue;
						E_OCPP1_Phase.L2N: fVoltageL2N := fValue;
						E_OCPP1_Phase.L3N: fVoltageL3N := fValue;
					ELSE
						mErrorValue := mValue;
					END_CASE
					IF fVoltageL1N >= 0 AND fVoltageL2N >= 0 AND fVoltageL3N >= 0 THEN
						fVoltage := (fVoltageL1N + fVoltageL2N + fVoltageL3N) * cfOneThird;
					END_IF
				END_IF
			ELSE
				mErrorValue := mValue;
			END_IF
	ELSE
		mErrorValue := mValue;
	END_CASE
END_IF
END_METHOD

END_FUNCTION_BLOCK

// ---- POUs/Helper/F_ChargePointStatusToString.TcPOU
FUNCTION F_ChargePointStatusToString : STRING(31)
VAR_INPUT
	eStatus : E_OCPP1_ChargePointStatus;
END_VAR

CASE eStatus OF
	E_OCPP1_ChargePointStatus.Available: F_ChargePointStatusToString := 'Available';
	E_OCPP1_ChargePointStatus.Preparing: F_ChargePointStatusToString := 'Preparing';
	E_OCPP1_ChargePointStatus.Charging: F_ChargePointStatusToString := 'Charging';
	E_OCPP1_ChargePointStatus.SuspendedEVSE: F_ChargePointStatusToString := 'SuspendedEVSE';
	E_OCPP1_ChargePointStatus.SuspendedEV: F_ChargePointStatusToString := 'SuspendedEV';
	E_OCPP1_ChargePointStatus.Finishing: F_ChargePointStatusToString := 'Finishing';
	E_OCPP1_ChargePointStatus.Reserved: F_ChargePointStatusToString := 'Reserved';
	E_OCPP1_ChargePointStatus.Unavailable: F_ChargePointStatusToString := 'Unavailable';
	E_OCPP1_ChargePointStatus.Faulted: F_ChargePointStatusToString := 'Faulted';
END_CASE

END_FUNCTION

// ---- POUs/Helper/F_TimeFromString.TcPOU
FUNCTION F_TimeFromString : LINT
VAR_INPUT
	sTime : STRING(31);
END_VAR

F_TimeFromString :=  ULINT_TO_LINT(DCTIME64_TO_FILETIME64(STRING_TO_DCTIME64(sTime)));

END_FUNCTION

// ---- GlobalTextList.TcGTLO
TEXTLIST GlobalTextList
  692 = '%'
  997 = '%.2f'
  842 = '%d'
  923 = '%f'
  777 = '%f.2'
  824 = '%s'
  404 = '...'
  358 = 'ChargePointStatus'
  204 = 'ChargingStation01'
  782 = 'ChargingStation02'
  333 = 'Charpoint Status'
  763 = 'Checkbox'
  265 = 'Conn1 '
  909 = 'Conn2'
  599 = 'Connected'
  5 = 'Connecting ...'
  614 = 'Connector 1'
  594 = 'Connector 2'
  379 = 'Connector2'
  153 = 'CS 01'
  39 = 'Current L1'
  882 = 'Current L1 [A]'
  351 = 'Current L2'
  356 = 'Current L2 [A]'
  377 = 'Current L3'
  166 = 'Current L3 [A]'
  274 = 'Energy Meter'
  756 = 'Energy Meter [kWh]'
  324 = 'EnergyActiveImport'
  10 = 'EVSE'
  122 = 'EVSE Connector'
  966 = 'EVSE Connector %d'
  366 = 'fbStation01.FB_Init.sIdent'
  334 = 'GetCompositeSchedule'
  762 = 'GroupBox'
  734 = 'kWh'
  860 = 'MeterStart'
  371 = 'MeterStart [Wh]'
  822 = 'MeterStop'
  362 = 'MeterStop  [Wh]'
  78 = 'MeterStop [Wh]'
  543 = 'nReservationId'
  184 = 'nStartTime'
  426 = 'nStopTime'
  232 = 'nTransactionId'
  695 = 'Power Active Importet'
  653 = 'Power Active Importet [kW]'
  146 = 'RemoteStart'
  816 = 'RemoteStop'
  969 = 'sAuthorizationStatus'
  761 = 'sChargePointModel'
  172 = 'sChargePointVendor'
  42 = 'sIdTag'
  759 = 'sIdTag / AuthStatus'
  88 = 'SoC'
  868 = 'Stations'
  476 = 'Voltage L1'
  551 = 'Voltage L1 [V]'
  579 = 'Voltage L2'
  4 = 'Voltage L2 [V]'
  344 = 'Voltage L3'
  696 = 'Voltage L3 [V]'
END_TEXTLIST

// ---- VISUs/Main_Visu.TcVIS
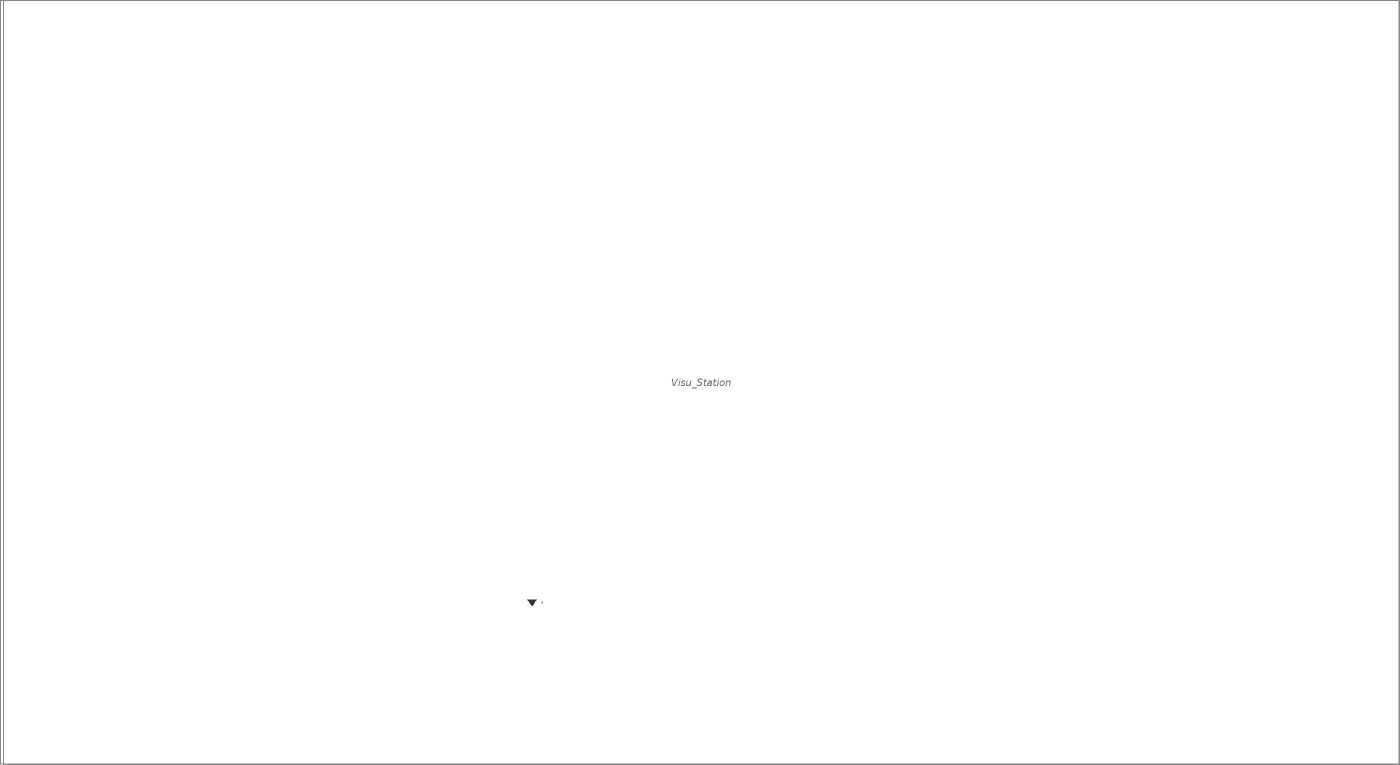
VISUALIZATION Main_Visu  // 1453x794
    SpinControl (562,625 1x0)
    TabControl (3,0 1450x794)
        shows Visu_Station(fbStation := MAIN.fbStation01)
        shows Visu_Station(fbStation := MAIN.fbStation02)
        [0]: TabTitle=ChargingStation01
        [1]: TabTitle=ChargingStation02
END_VISUALIZATION

// ---- VISUs/Measurand.TcVIS
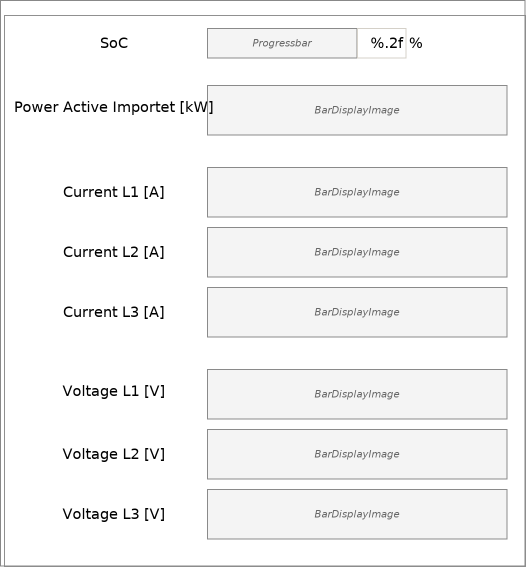
VISUALIZATION Measurand  // 526x567
VAR_IN_OUT
	fbMeasurand : FB_SampledValueMeasurands; 
END_VAR
    GroupBox (4,7 522x560)
        BarDisplayImage (203,160 300x50), value: fbMeasurand.fCurrentImportL1, style: BarDisplayImage-Gray, scale format: %.1f, scale 0..32
        Progressbar (203,21 150x30), variable: fbMeasurand.fStateOfCharge
        Textfield (353,21 49x30), "%.2f", text variable: fbMeasurand.fStateOfCharge
        Label (35,160 150x50), "Current L1 [A]"
        Label (35,220 150x50), "Current L2 [A]"
        Label (35,280 150x50), "Current L3 [A]"
        BarDisplayImage (203,362 300x50), value: fbMeasurand.fVoltageL1N, style: BarDisplayImage-Gray, scale format: %.1f, scale 0..250
        Label (35,362 150x44), "Voltage L1 [V]"
        Label (35,422 150x50), "Voltage L2 [V]"
        Label (35,482 150x50), "Voltage L3 [V]"
        Label (35,21 150x30), "SoC"
        BarDisplayImage (203,78 300x50), value: fbMeasurand.fPowerActiveImport, style: BarDisplayImage-Gray, scale format: %.1f, scale 0..22
        Label (35,85 150x30), "Power Active Importet [kW]"
        BarDisplayImage (203,220 300x50), value: fbMeasurand.fCurrentImportL2, style: BarDisplayImage-Gray, scale format: %.1f, scale 0..32
        BarDisplayImage (203,280 300x50), value: fbMeasurand.fCurrentImportL3, style: BarDisplayImage-Gray, scale format: %.1f, scale 0..32
        BarDisplayImage (203,422 300x50), value: fbMeasurand.fVoltageL2N, style: BarDisplayImage-Gray, scale format: %.1f, scale 0..250
        BarDisplayImage (203,482 300x50), value: fbMeasurand.fVoltageL3N, style: BarDisplayImage-Gray, scale format: %.1f, scale 0..250
        Label (402,21 47x30), "%"
END_VISUALIZATION

// ---- VISUs/Visu_BootNotification.TcVIS
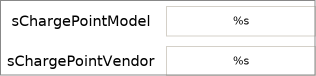
VISUALIZATION Visu_BootNotification  // 316x76
VAR_IN_OUT
	fbStation 		: FB_Station;
END_VAR
    Textfield (166,6 150x30), "%s", text variable: fbStation._stVisu.stBoot.sChargePointModel
    Textfield (166,46 150x30), "%s", text variable: fbStation._stVisu.stBoot.sChargePointVendor
    Label (6,6 150x30), "sChargePointModel"
    Label (6,46 150x30), "sChargePointVendor"
END_VISUALIZATION

// ---- VISUs/Visu_Connector.TcVIS
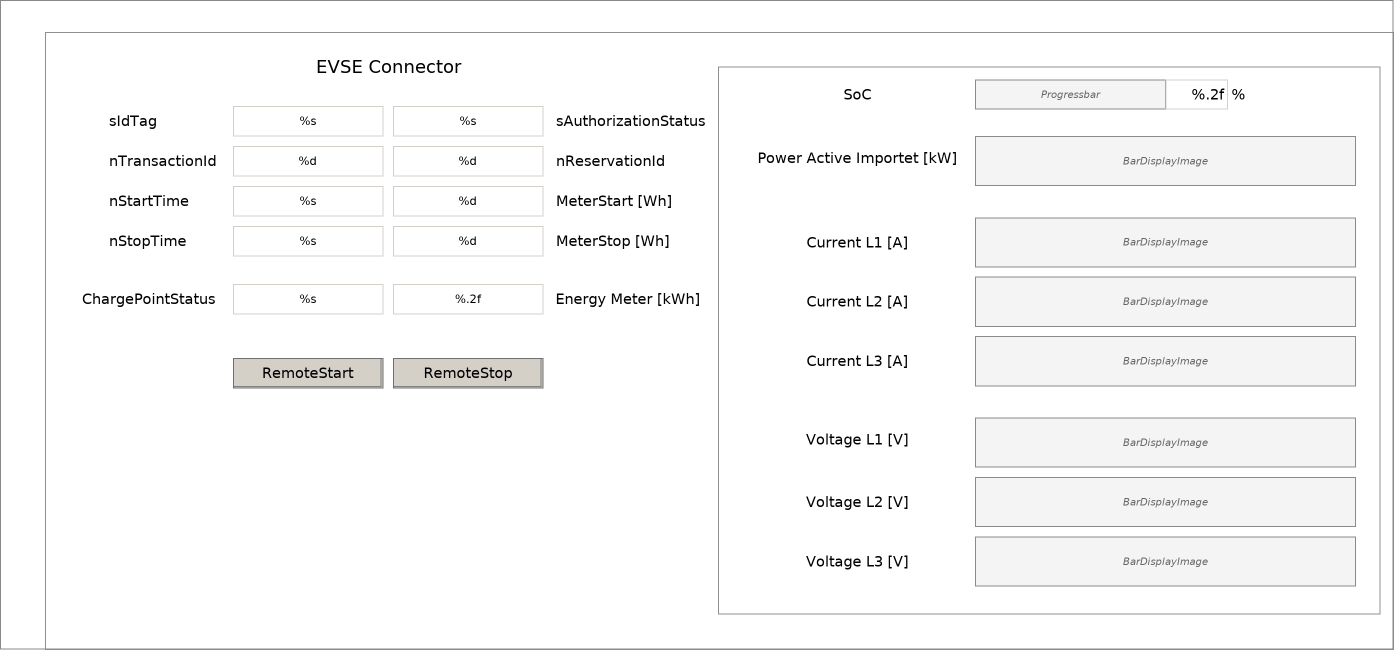
VISUALIZATION Visu_Connector  // 1394x650
VAR_IN_OUT
	stConnector : ST_Connector; 
 	fbMeasurand : FB_SampledValueMeasurands; 
	bRemoteStart : BOOL;
	bRemoteStop : BOOL; 
END_VAR
    GroupBox (45,24 1349x626)
        Textfield (188,82 150x30), "%s", text variable: stConnector.sIdTag
        Label (61,82 117x30), "sIdTag"
        Textfield (188,122 150x30), "%d", text variable: stConnector.nTransactionID
        Textfield (188,162 150x30), "%s", text variable: stConnector.sStartTime
        Textfield (188,202 150x30), "%s", text variable: stConnector.sStopTime
        Label (61,122 117x30), "nTransactionId"
        Label (61,162 117x30), "nStartTime"
        Label (61,202 117x30), "nStopTime"
        Textfield (348,82 150x30), "%s", text variable: stConnector.sAuthorizationStatus
        Textfield (188,260 150x30), "%s", text variable: stConnector.sChargpointStatus
        Label (29,260 150x30), "ChargePointStatus"
        Textfield (348,162 150x30), "%d", text variable: stConnector.nMeterStart
        Label (508,162 150x30), "MeterStart [Wh]"
        Textfield (348,202 150x30), "%d", text variable: stConnector.nMeterStop
        Label (508,202 150x30), "MeterStop [Wh]"
        Label (508,82 150x30), "sAuthorizationStatus"
        Textfield (348,122 150x30), "%d", text variable: stConnector.nReservationId
        Label (508,122 150x30), "nReservationId"
        Textfield (348,260 150x30), "%.2f", text variable: fbMeasurand.fEnergyActiveImportRegister
        Label (508,260 150x30), "Energy Meter [kWh]"
        Label (261,28 166x30), "EVSE Connector"
        Button (188,334 150x30), "RemoteStart"
            tap bRemoteStart
        Button (348,334 150x30), "RemoteStop"
            tap bRemoteStop
        Frame (668,28 667x562)
            shows Measurand(fbMeasurand := fbMeasurand)
END_VISUALIZATION

// ---- VISUs/Visu_Station.TcVIS
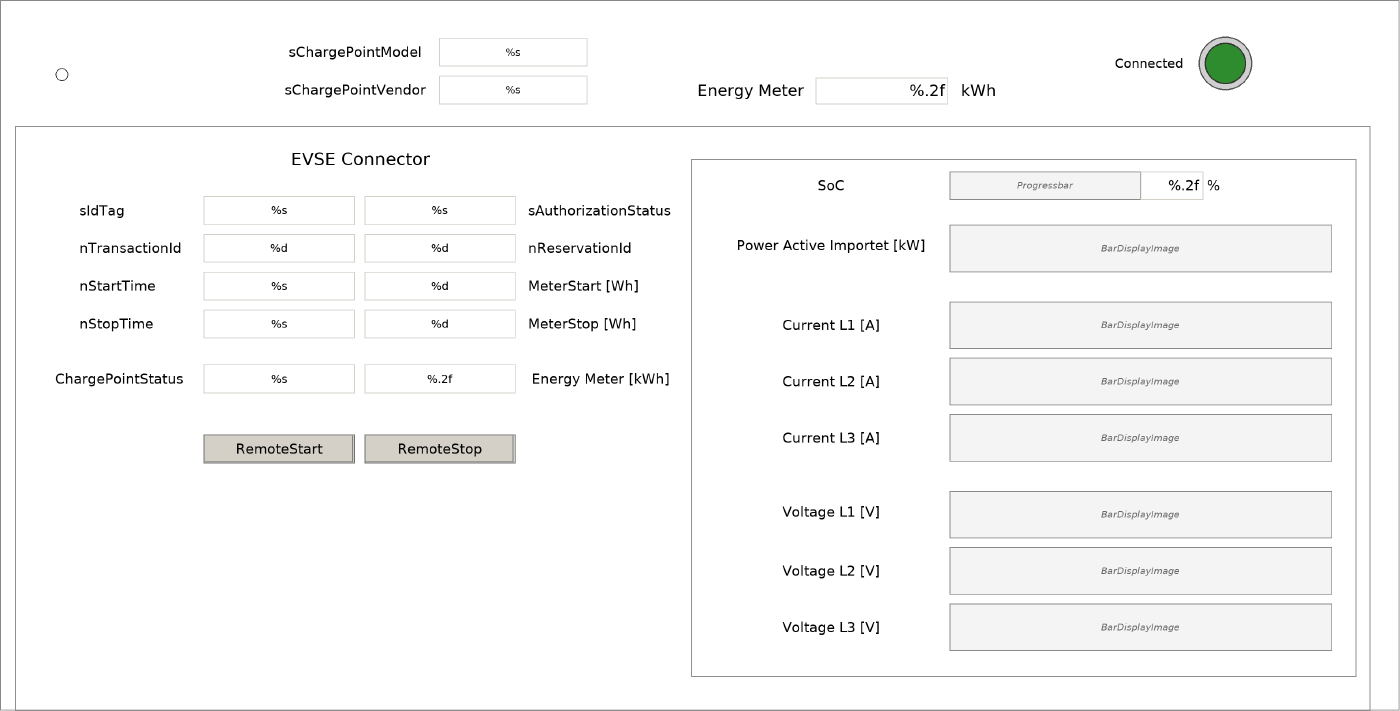
VISUALIZATION Visu_Station  // 1588x807
VAR_IN_OUT
	fbStation 		: FB_Station;
END_VAR
VAR 
	nConnectorVisu :UDINT; 
END_VAR
    Frame (-34,109 1588x698), frame switch variable: nConnectorVisu
        shows Visu_Connector(stConnector := fbStation._stVisu.aConnector[1], fbMeasurand := fbStation.arrMeasurands[1], bRemoteStart := fbStation._arrRemoteStart[1], bRemoteStop := fbStation._arrRemoteStop[1])
        shows Visu_Connector(stConnector := fbStation._stVisu.aConnector[2], fbMeasurand := fbStation.arrMeasurands[2], bRemoteStart := fbStation._arrRemoteStart[2], bRemoteStop := fbStation._arrRemoteStop[2])
    Frame (313,37 353x81)
        shows Visu_BootNotification(fbStation := fbStation)
    RadioButton (61,51 150x67), variable: nConnectorVisu
        Areas[0]: Text=Connector 1
        Areas[1]: Text=Connector 2
    Lamp1 (1355,37 70x70), variable: fbStation.bOpen, style: Lamp-Lamp1-Green
    Label (1184,37 161x70), "Connected"
    Textfield (925,88 150x30), "%.2f", text variable: fbStation.arrMeasurands[1].fEnergyActiveImportRegister + fbStation.arrMeasurands[2].fEnergyActiveImportRegister
    Label (765,88 150x30), "Energy Meter"
    Label (1079,88 62x30), "kWh"
END_VISUALIZATION
